{attribute 'qualified_only'}
VAR_GLOBAL CONSTANT
	fMaxTemperature : REAL := 80;
	fMaxLevelPercentage: REAL := 90.0;
	
	fRequiredTemperature: REAL := 50.0;
	fRequiredLevel : REAL := 30;
	
	fCoolingSpeed : REAL := 10;
	fTransferSpeed : REAL := 10;
	
	fProcessLevel : REAL := 10;
	fProcessTemperature : REAL := 5;
END_VAR

(* stored: Version 1.1.0.1, ProductVersion 3.1.4024.16
   GVL GVL: Id {2fb9fffc-91f2-4040-b4c7-3f897fd92de1} *)
